{attribute addProperty BoxType "EJ2522-0000-0022"}
{attribute addProperty Id "ControlAT %Q*Control_A1EB0E501621Frequency_valueAT %Q*UINT16217"}
{attribute addProperty CRC "174198979"}
{attribute addProperty SizeInBites "32"}
{attribute addProperty SizeInBytes "4"}
TYPE PTO_Control_Channel_0A6210C3 :
STRUCT
	{attribute addProperty Name "Control"}
	Control AT %Q* : Control_A1EB0E50;
	{attribute addProperty Name "Frequency_value"}
	Frequency_value AT %Q* : UINT;
END_STRUCT
END_TYPE

(* stored: Version 1.2.0.0, ProductVersion 3.1.4024.9
   DUT PTO_Control_Channel_0A6210C3: Id {9b9a0093-a600-4794-ac75-fac3170684d0} *)
